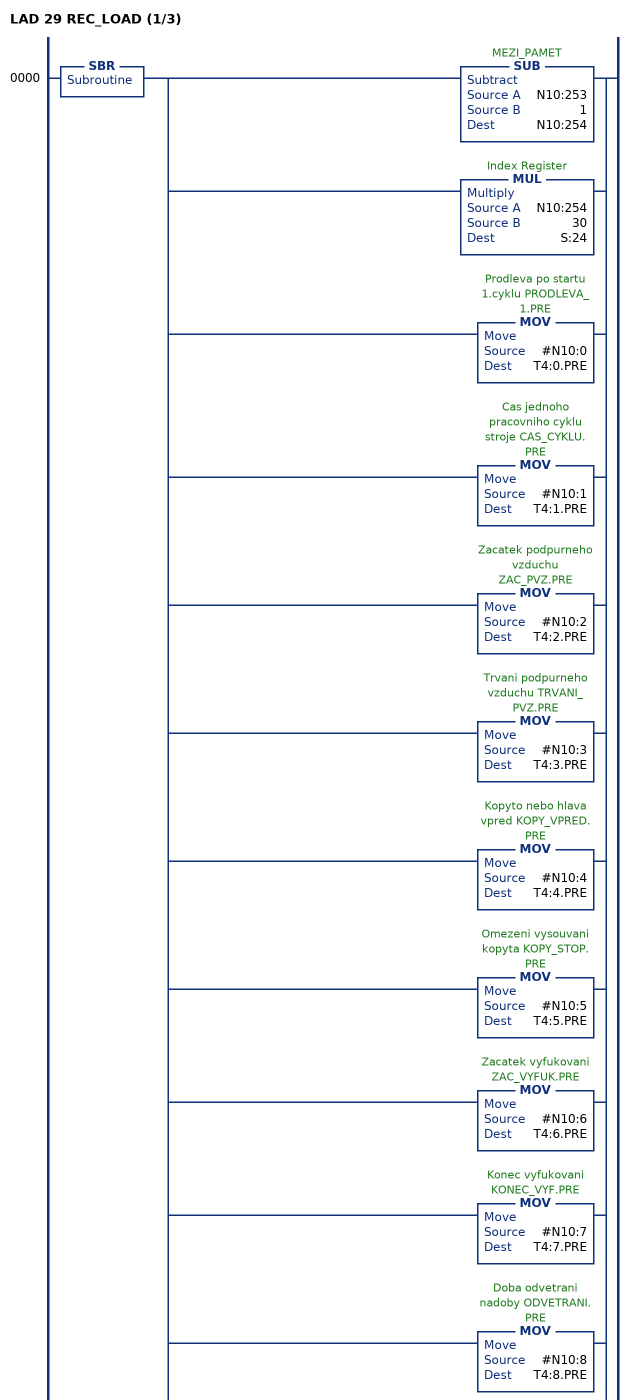
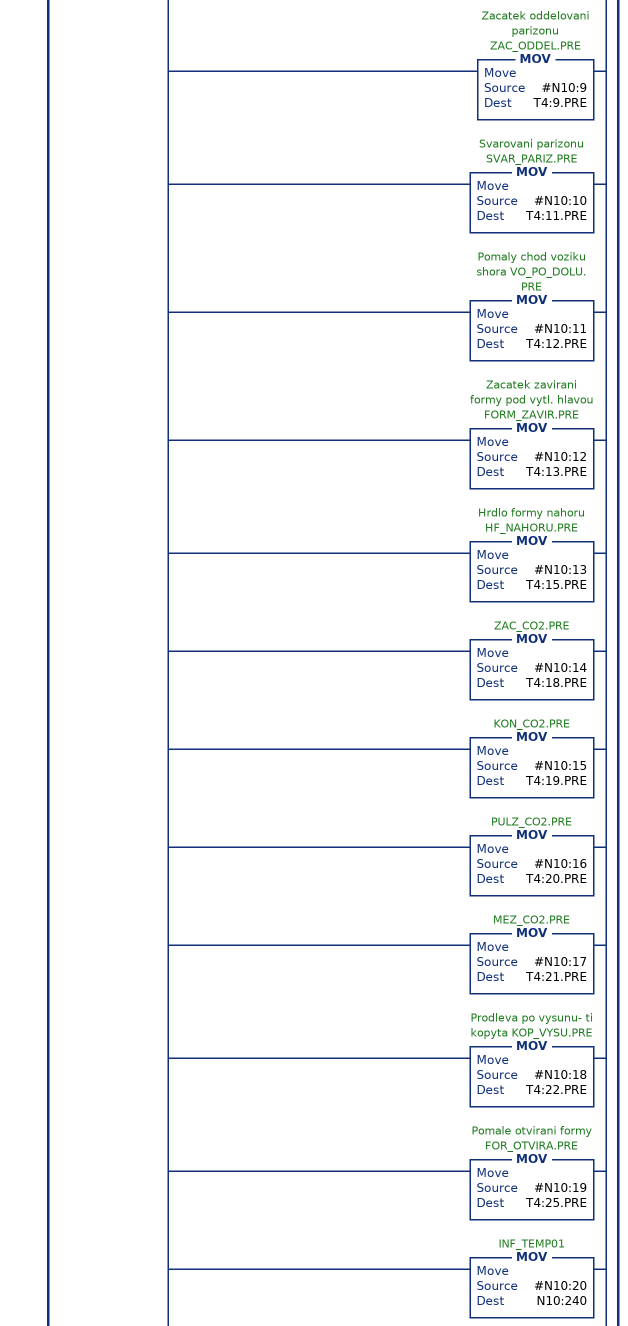
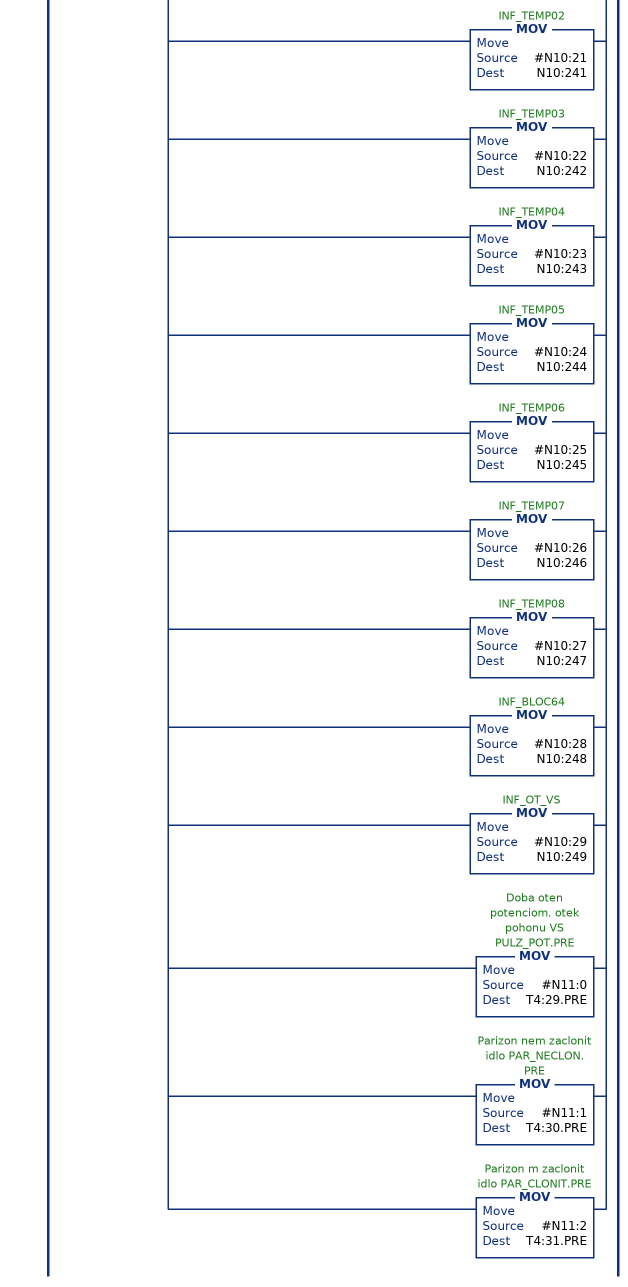
% Rung: 0 %
SOR SBR BST SUB N10:253 1 N10:254 NXB MUL N10:254 30 S:24 NXB MOV #N10:0 T4:0.PRE NXB MOV #N10:1 T4:1.PRE NXB MOV #N10:2 T4:2.PRE NXB MOV #N10:3 T4:3.PRE NXB MOV #N10:4 T4:4.PRE NXB MOV #N10:5 T4:5.PRE NXB MOV #N10:6 T4:6.PRE NXB MOV #N10:7 T4:7.PRE NXB MOV #N10:8 T4:8.PRE NXB MOV #N10:9 T4:9.PRE NXB MOV #N10:10 T4:11.PRE NXB MOV #N10:11 T4:12.PRE NXB MOV #N10:12 T4:13.PRE NXB MOV #N10:13 T4:15.PRE NXB MOV #N10:14 T4:18.PRE NXB MOV #N10:15 T4:19.PRE NXB MOV #N10:16 T4:20.PRE NXB MOV #N10:17 T4:21.PRE NXB MOV #N10:18 T4:22.PRE NXB MOV #N10:19 T4:25.PRE NXB MOV #N10:20 N10:240 NXB MOV #N10:21 N10:241 NXB MOV #N10:22 N10:242 NXB MOV #N10:23 N10:243 NXB MOV #N10:24 N10:244 NXB MOV #N10:25 N10:245 NXB MOV #N10:26 N10:246 NXB MOV #N10:27 N10:247 NXB MOV #N10:28 N10:248 NXB MOV #N10:29 N10:249 NXB MOV #N11:0 T4:29.PRE NXB MOV #N11:1 T4:30.PRE NXB MOV #N11:2 T4:31.PRE BND EOR
%   N10:253  REC_NO_PAR %
%   N10:254  MEZI_PAMET %
%   S:24  "Index Register" %
%   N10:0  REC_WORD00 %
%   T4:0  PRODLEVA_1  "Prodleva po startu 1.cyklu" %
%   N10:1  REC_WORD01 %
%   T4:1  CAS_CYKLU  "Cas jednoho pracovniho cyklu stroje" %
%   N10:2  REC_WORD02 %
%   T4:2  ZAC_PVZ  "Zacatek podpurneho vzduchu" %
%   N10:3  REC_WORD03 %
%   T4:3  TRVANI_PVZ  "Trvani podpurneho vzduchu" %
%   N10:4  REC_WORD04 %
%   T4:4  KOPY_VPRED  "Kopyto nebo hlava vpred" %
%   N10:5  REC_WORD05 %
%   T4:5  KOPY_STOP  "Omezeni vysouvani kopyta" %
%   N10:6  REC_WORD06 %
%   T4:6  ZAC_VYFUK  "Zacatek vyfukovani" %
%   N10:7  REC_WORD07 %
%   T4:7  KONEC_VYF  "Konec vyfukovani" %
%   N10:8  REC_WORD08 %
%   T4:8  ODVETRANI  "Doba odvetrani nadoby" %
%   N10:9  REC_WORD09 %
%   T4:9  ZAC_ODDEL  "Zacatek oddelovani parizonu" %
%   N10:10  REC_WORD10 %
%   T4:11  SVAR_PARIZ  "Svarovani parizonu" %
%   N10:11  REC_WORD11 %
%   T4:12  VO_PO_DOLU  "Pomaly chod voziku shora" %
%   N10:12  REC_WORD12 %
%   T4:13  FORM_ZAVIR  "Zacatek zavirani formy pod vytl. hlavou" %
%   N10:13  REC_WORD13 %
%   T4:15  HF_NAHORU  "Hrdlo formy nahoru" %
%   N10:14  REC_WORD14 %
%   T4:18  ZAC_CO2 %
%   N10:15  REC_WORD15 %
%   T4:19  KON_CO2 %
%   N10:16  REC_WORD16 %
%   T4:20  PULZ_CO2 %
%   N10:17  REC_WORD17 %
%   T4:21  MEZ_CO2 %
%   N10:18  REC_WORD18 %
%   T4:22  KOP_VYSU  "Prodleva po vysunu- ti kopyta" %
%   N10:19  REC_WORD19 %
%   T4:25  FOR_OTVIRA  "Pomale otvirani formy" %
%   N10:20  REC_WORD20 %
%   N10:240  INF_TEMP01 %
%   N10:21  REC_WORD21 %
%   N10:241  INF_TEMP02 %
%   N10:22  REC_WORD22 %
%   N10:242  INF_TEMP03 %
%   N10:23  REC_WORD23 %
%   N10:243  INF_TEMP04 %
%   N10:24  REC_WORD24 %
%   N10:244  INF_TEMP05 %
%   N10:25  REC_WORD25 %
%   N10:245  INF_TEMP06 %
%   N10:26  REC_WORD26 %
%   N10:246  INF_TEMP07 %
%   N10:27  REC_WORD27 %
%   N10:247  INF_TEMP08 %
%   N10:28  REC_WORD28 %
%   N10:248  INF_BLOC64 %
%   N10:29  REC_WORD29 %
%   N10:249  INF_OT_VS %
%   N11:0  REC_WORD30 %
%   T4:29  PULZ_POT  "Doba oten potenciom. otek pohonu VS" %
%   N11:1  REC_WORD31 %
%   T4:30  PAR_NECLON  "Parizon nem zaclonit idlo" %
%   N11:2  REC_WORD32 %
%   T4:31  PAR_CLONIT  "Parizon m zaclonit idlo" %

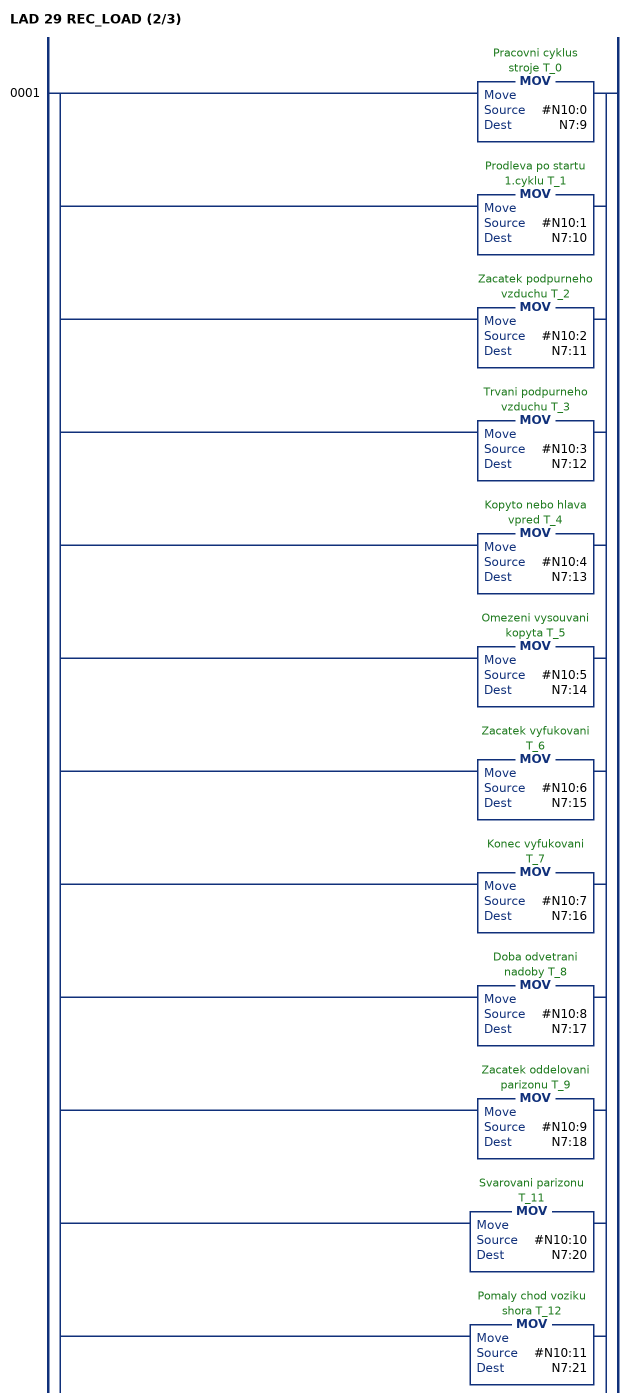

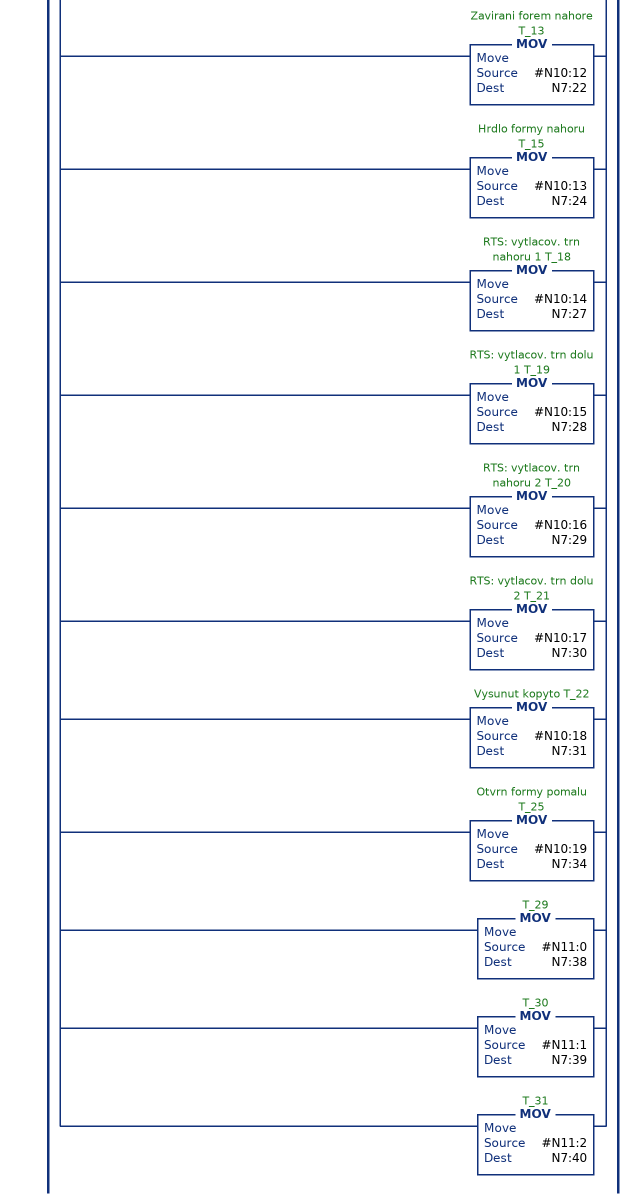
% Rung: 1 %
SOR BST MOV #N10:0 N7:9 NXB MOV #N10:1 N7:10 NXB MOV #N10:2 N7:11 NXB MOV #N10:3 N7:12 NXB MOV #N10:4 N7:13 NXB MOV #N10:5 N7:14 NXB MOV #N10:6 N7:15 NXB MOV #N10:7 N7:16 NXB MOV #N10:8 N7:17 NXB MOV #N10:9 N7:18 NXB MOV #N10:10 N7:20 NXB MOV #N10:11 N7:21 NXB MOV #N10:12 N7:22 NXB MOV #N10:13 N7:24 NXB MOV #N10:14 N7:27 NXB MOV #N10:15 N7:28 NXB MOV #N10:16 N7:29 NXB MOV #N10:17 N7:30 NXB MOV #N10:18 N7:31 NXB MOV #N10:19 N7:34 NXB MOV #N11:0 N7:38 NXB MOV #N11:1 N7:39 NXB MOV #N11:2 N7:40 BND EOR
%   N10:0  REC_WORD00 %
%   N7:9  T_0  "Pracovni cyklus stroje" %
%   N10:1  REC_WORD01 %
%   N7:10  T_1  "Prodleva po startu 1.cyklu" %
%   N10:2  REC_WORD02 %
%   N7:11  T_2  "Zacatek podpurneho vzduchu" %
%   N10:3  REC_WORD03 %
%   N7:12  T_3  "Trvani podpurneho vzduchu" %
%   N10:4  REC_WORD04 %
%   N7:13  T_4  "Kopyto nebo hlava vpred" %
%   N10:5  REC_WORD05 %
%   N7:14  T_5  "Omezeni vysouvani kopyta" %
%   N10:6  REC_WORD06 %
%   N7:15  T_6  "Zacatek vyfukovani" %
%   N10:7  REC_WORD07 %
%   N7:16  T_7  "Konec vyfukovani" %
%   N10:8  REC_WORD08 %
%   N7:17  T_8  "Doba odvetrani nadoby" %
%   N10:9  REC_WORD09 %
%   N7:18  T_9  "Zacatek oddelovani parizonu" %
%   N10:10  REC_WORD10 %
%   N7:20  T_11  "Svarovani parizonu" %
%   N10:11  REC_WORD11 %
%   N7:21  T_12  "Pomaly chod voziku shora" %
%   N10:12  REC_WORD12 %
%   N7:22  T_13  "Zavirani forem nahore" %
%   N10:13  REC_WORD13 %
%   N7:24  T_15  "Hrdlo formy nahoru" %
%   N10:14  REC_WORD14 %
%   N7:27  T_18  "RTS: vytlacov. trn nahoru 1" %
%   N10:15  REC_WORD15 %
%   N7:28  T_19  "RTS: vytlacov. trn dolu 1" %
%   N10:16  REC_WORD16 %
%   N7:29  T_20  "RTS: vytlacov. trn nahoru 2" %
%   N10:17  REC_WORD17 %
%   N7:30  T_21  "RTS: vytlacov. trn dolu 2" %
%   N10:18  REC_WORD18 %
%   N7:31  T_22  "Vysunut kopyto" %
%   N10:19  REC_WORD19 %
%   N7:34  T_25  "Otvrn formy pomalu" %
%   N11:0  REC_WORD30 %
%   N7:38  T_29 %
%   N11:1  REC_WORD31 %
%   N7:39  T_30 %
%   N11:2  REC_WORD32 %
%   N7:40  T_31 %

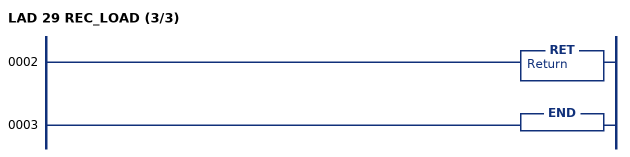
% Rung: 2 %
SOR RET EOR
% Rung: 3 %
SOR END EOR

LADDER 30 "REG_TEPLOT"
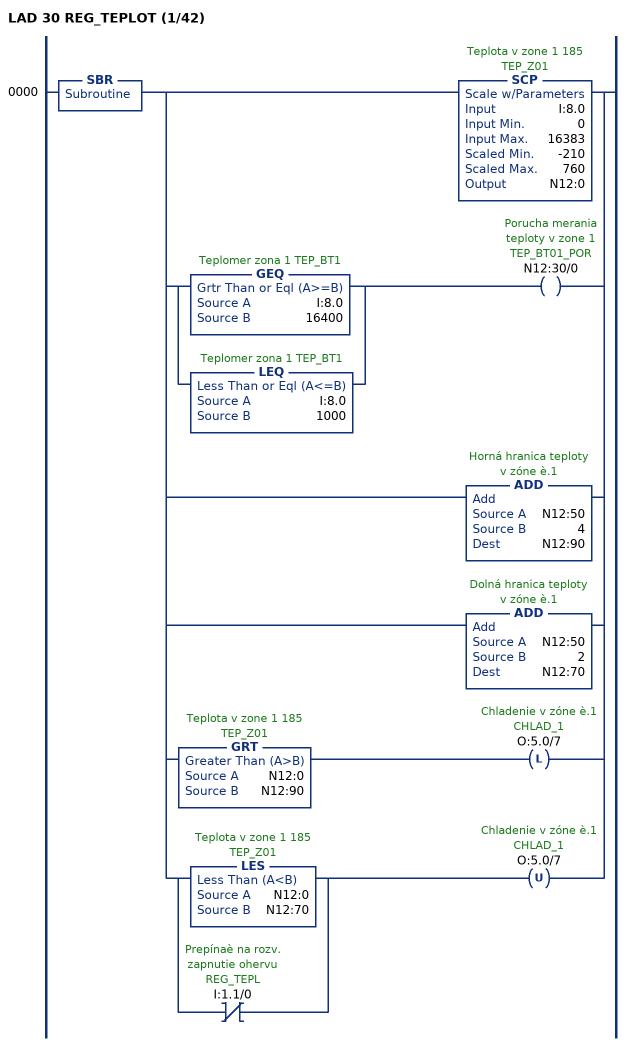
% Rung: 0 %
SOR SBR BST SCP I:8.0 0 16383 -210 760 N12:0 NXB BST GEQ I:8.0 16400 NXB LEQ I:8.0 1000 BND OTE N12:30/0 NXB ADD N12:50 4 N12:90 NXB ADD N12:50 2 N12:70 NXB GRT N12:0 N12:90 OTL O:5.0/7 NXB BST LES N12:0 N12:70 NXB XIO I:1.1/0 BND OTU O:5.0/7 BND EOR
%   I:8.0  TEP_BT1  "Teplomer zona 1" %
%   N12:0  TEP_Z01  "Teplota v zone 1 185" %
%   N12:30/0  TEP_BT01_POR  "Porucha merania teploty v zone 1" %
%   N12:50  "Žiadaná teplota v zóne è.1" %
%   N12:90  "Horná hranica teploty v zóne è.1" %
%   N12:70  "Dolná hranica teploty v zóne è.1" %
%   O:5.0/7  CHLAD_1  "Chladenie v zóne è.1" %
%   I:1.1/0  REG_TEPL  "Prepínaè na rozv. zapnutie ohervu" %

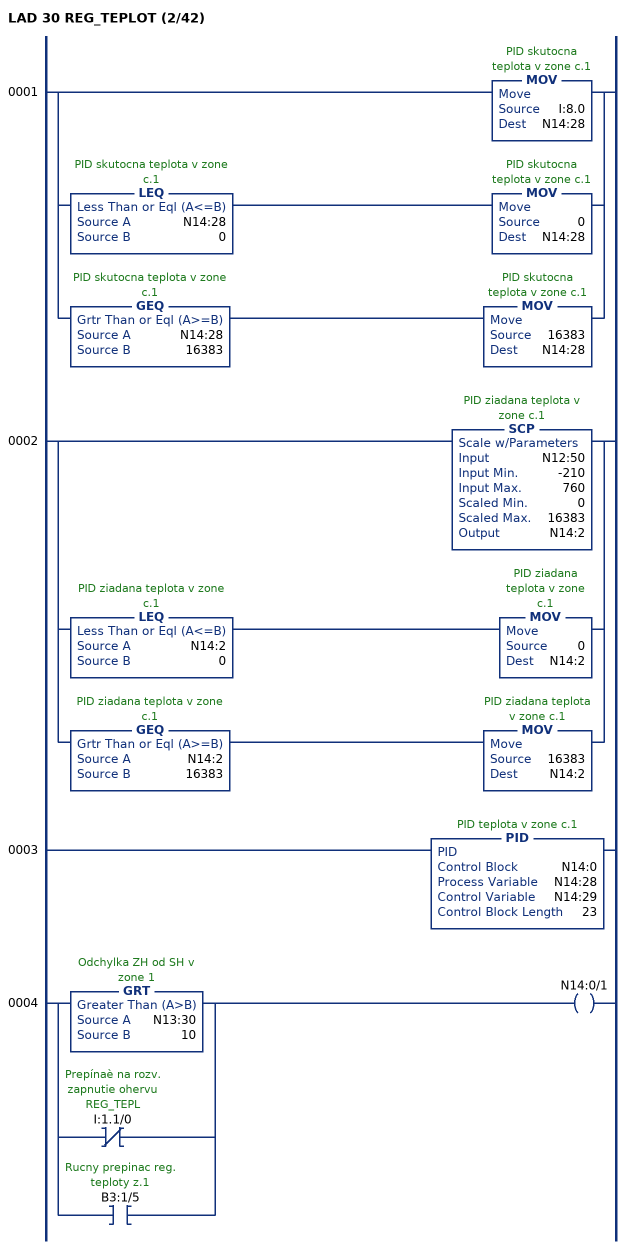
% Rung: 1 %
SOR BST MOV I:8.0 N14:28 NXB LEQ N14:28 0 MOV 0 N14:28 NXB GEQ N14:28 16383 MOV 16383 N14:28 BND EOR
%   I:8.0  TEP_BT1  "Teplomer zona 1" %
%   N14:28  "PID skutocna teplota v zone c.1" %
% Rung: 2 %
SOR BST SCP N12:50 -210 760 0 16383 N14:2 NXB LEQ N14:2 0 MOV 0 N14:2 NXB GEQ N14:2 16383 MOV 16383 N14:2 BND EOR
%   N12:50  "Žiadaná teplota v zóne è.1" %
%   N14:2  "PID ziadana teplota v zone c.1" %
% Rung: 3 %
SOR PID N14:0 N14:28 N14:29 23 EOR
%   N14:0  "PID teplota v zone c.1" %
%   N14:28  "PID skutocna teplota v zone c.1" %
% Rung: 4 %
SOR BST GRT N13:30 10 NXB XIO I:1.1/0 NXB XIC B3:1/5 BND OTE N14:0/1 EOR
%   N13:30  "Odchylka ZH od SH v zone 1" %
%   I:1.1/0  REG_TEPL  "Prepínaè na rozv. zapnutie ohervu" %
%   B3:1/5  "Rucny prepinac reg. teploty z.1" %

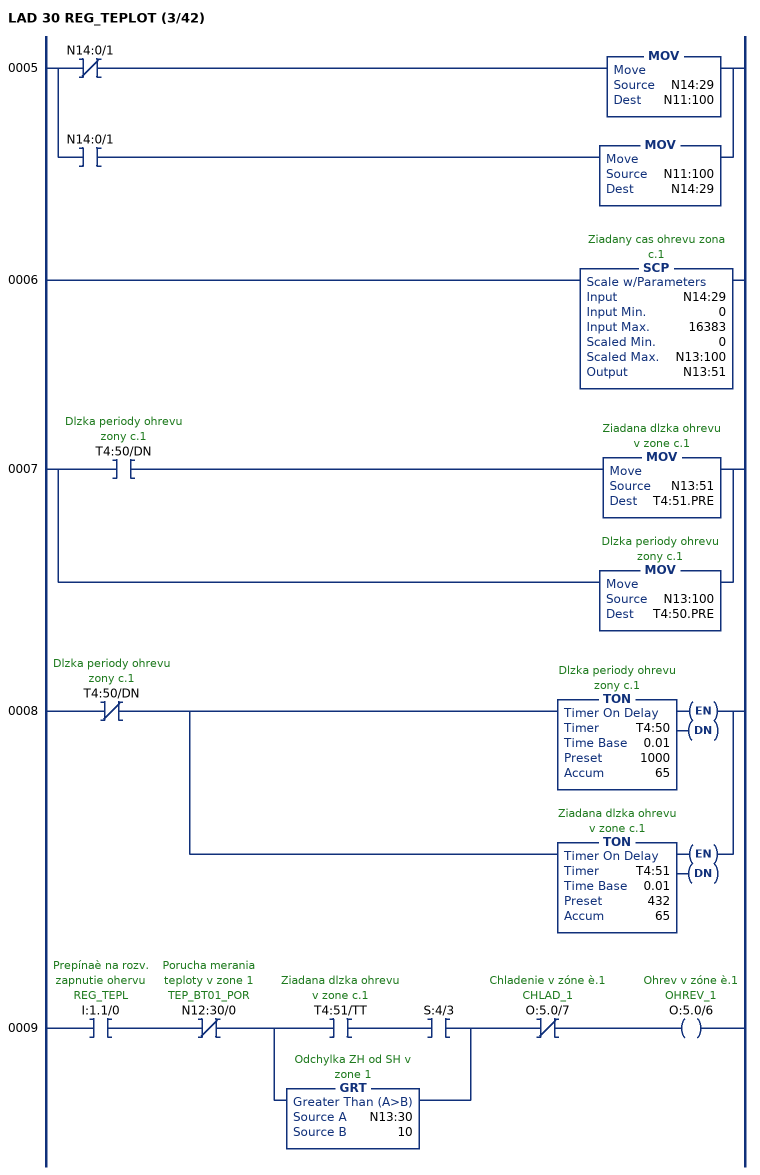
% Rung: 5 %
SOR BST XIO N14:0/1 MOV N14:29 N11:100 NXB XIC N14:0/1 MOV N11:100 N14:29 BND EOR
% Rung: 6 %
SOR SCP N14:29 0 16383 0 N13:100 N13:51 EOR
%   N13:51  "Ziadany cas ohrevu zona c.1" %
% Rung: 7 %
SOR BST XIC T4:50/DN MOV N13:51 T4:51.PRE NXB MOV N13:100 T4:50.PRE BND EOR
%   T4:50  "Dlzka periody ohrevu zony c.1" %
%   N13:51  "Ziadany cas ohrevu zona c.1" %
%   T4:51  "Ziadana dlzka ohrevu v zone c.1" %
% Rung: 8 %
SOR XIO T4:50/DN BST TON T4:50 0.01 1000 65 NXB TON T4:51 0.01 432 65 BND EOR
%   T4:50  "Dlzka periody ohrevu zony c.1" %
%   T4:51  "Ziadana dlzka ohrevu v zone c.1" %
% Rung: 9 %
SOR XIC I:1.1/0 XIO N12:30/0 BST XIC T4:51/TT XIC S:4/3 NXB GRT N13:30 10 BND XIO O:5.0/7 OTE O:5.0/6 EOR
%   I:1.1/0  REG_TEPL  "Prepínaè na rozv. zapnutie ohervu" %
%   N12:30/0  TEP_BT01_POR  "Porucha merania teploty v zone 1" %
%   T4:51  "Ziadana dlzka ohrevu v zone c.1" %
%   N13:30  "Odchylka ZH od SH v zone 1" %
%   O:5.0/7  CHLAD_1  "Chladenie v zóne è.1" %
%   O:5.0/6  OHREV_1  "Ohrev v zóne è.1" %

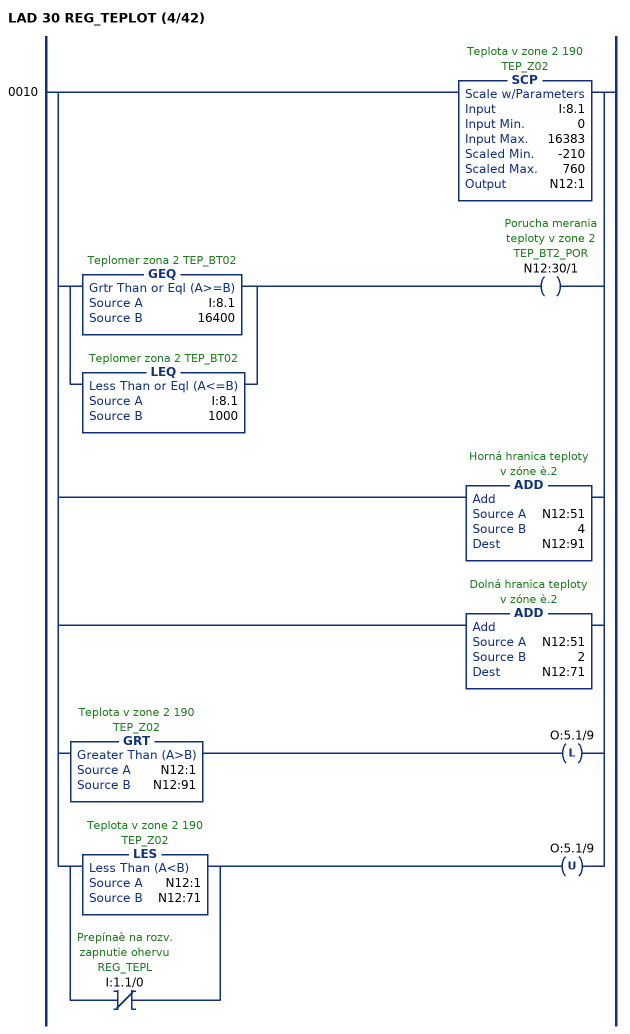
% Rung: 10 %
SOR BST SCP I:8.1 0 16383 -210 760 N12:1 NXB BST GEQ I:8.1 16400 NXB LEQ I:8.1 1000 BND OTE N12:30/1 NXB ADD N12:51 4 N12:91 NXB ADD N12:51 2 N12:71 NXB GRT N12:1 N12:91 OTL O:5.1/9 NXB BST LES N12:1 N12:71 NXB XIO I:1.1/0 BND OTU O:5.1/9 BND EOR
%   I:8.1  TEP_BT02  "Teplomer zona 2" %
%   N12:1  TEP_Z02  "Teplota v zone 2 190" %
%   N12:30/1  TEP_BT2_POR  "Porucha merania teploty v zone 2" %
%   N12:51  "Žiadaná teplota v zóne è.2" %
%   N12:91  "Horná hranica teploty v zóne è.2" %
%   N12:71  "Dolná hranica teploty v zóne è.2" %
%   I:1.1/0  REG_TEPL  "Prepínaè na rozv. zapnutie ohervu" %

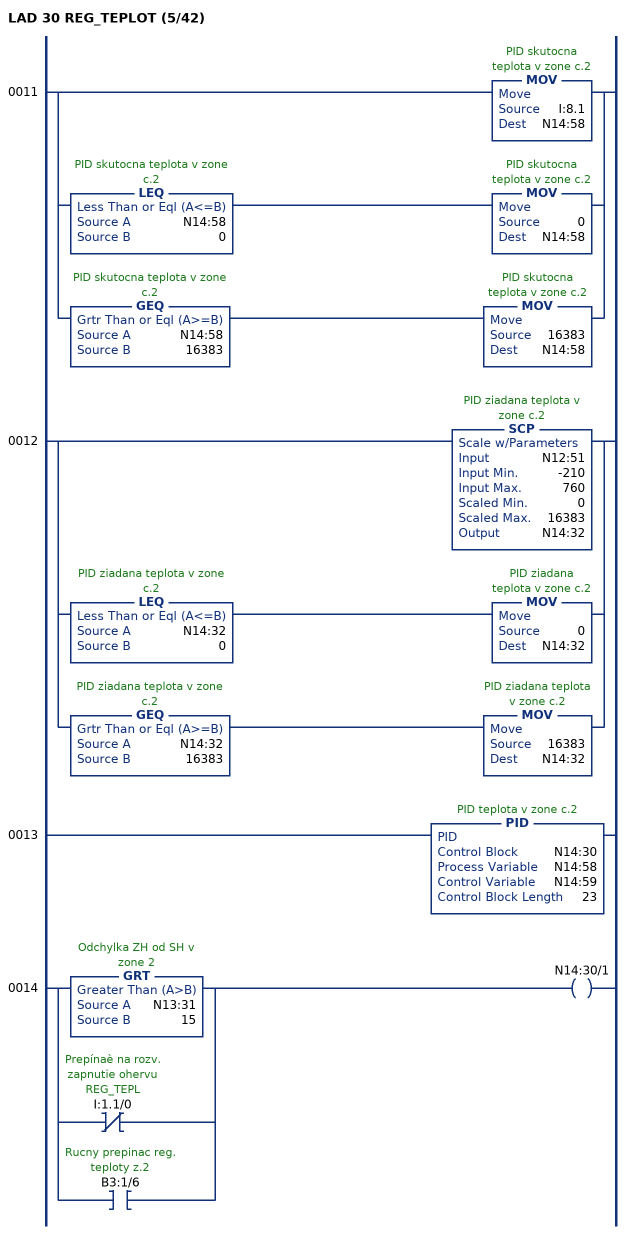
% Rung: 11 %
SOR BST MOV I:8.1 N14:58 NXB LEQ N14:58 0 MOV 0 N14:58 NXB GEQ N14:58 16383 MOV 16383 N14:58 BND EOR
%   I:8.1  TEP_BT02  "Teplomer zona 2" %
%   N14:58  "PID skutocna teplota v zone c.2" %
% Rung: 12 %
SOR BST SCP N12:51 -210 760 0 16383 N14:32 NXB LEQ N14:32 0 MOV 0 N14:32 NXB GEQ N14:32 16383 MOV 16383 N14:32 BND EOR
%   N12:51  "Žiadaná teplota v zóne è.2" %
%   N14:32  "PID ziadana teplota v zone c.2" %
% Rung: 13 %
SOR PID N14:30 N14:58 N14:59 23 EOR
%   N14:30  "PID teplota v zone c.2" %
%   N14:58  "PID skutocna teplota v zone c.2" %
% Rung: 14 %
SOR BST GRT N13:31 15 NXB XIO I:1.1/0 NXB XIC B3:1/6 BND OTE N14:30/1 EOR
%   N13:31  "Odchylka ZH od SH v zone 2" %
%   I:1.1/0  REG_TEPL  "Prepínaè na rozv. zapnutie ohervu" %
%   B3:1/6  "Rucny prepinac reg. teploty z.2" %

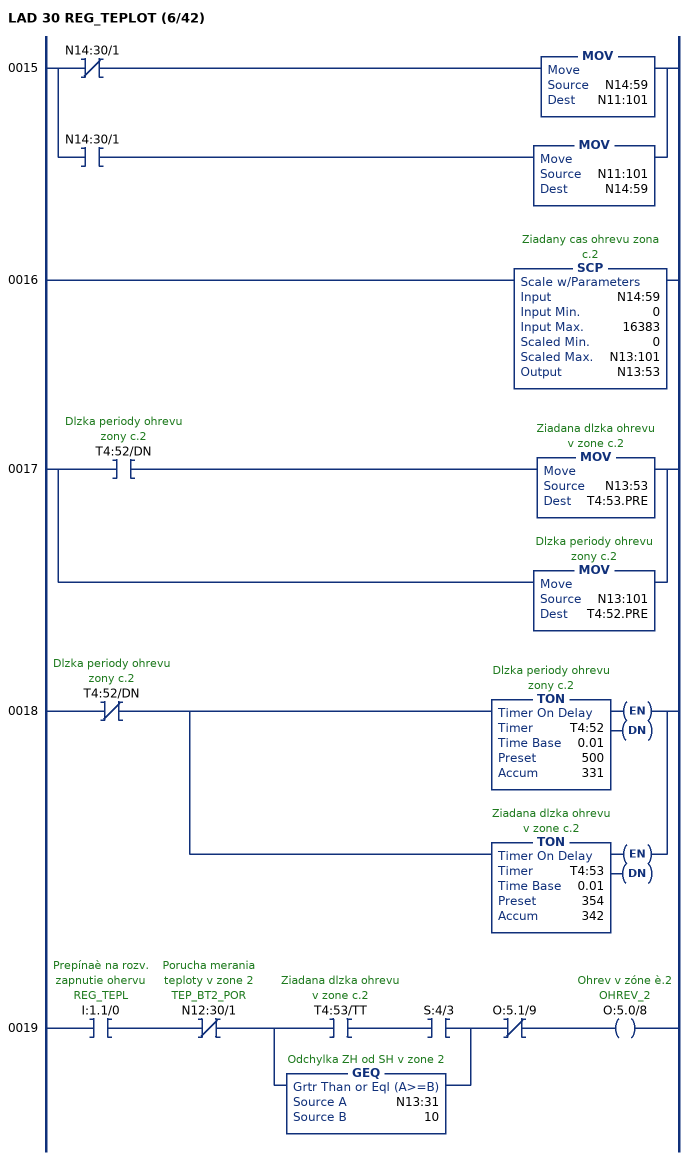
% Rung: 15 %
SOR BST XIO N14:30/1 MOV N14:59 N11:101 NXB XIC N14:30/1 MOV N11:101 N14:59 BND EOR
% Rung: 16 %
SOR SCP N14:59 0 16383 0 N13:101 N13:53 EOR
%   N13:53  "Ziadany cas ohrevu zona c.2" %
% Rung: 17 %
SOR BST XIC T4:52/DN MOV N13:53 T4:53.PRE NXB MOV N13:101 T4:52.PRE BND EOR
%   T4:52  "Dlzka periody ohrevu zony c.2" %
%   N13:53  "Ziadany cas ohrevu zona c.2" %
%   T4:53  "Ziadana dlzka ohrevu v zone c.2" %
% Rung: 18 %
SOR XIO T4:52/DN BST TON T4:52 0.01 500 331 NXB TON T4:53 0.01 354 342 BND EOR
%   T4:52  "Dlzka periody ohrevu zony c.2" %
%   T4:53  "Ziadana dlzka ohrevu v zone c.2" %
% Rung: 19 %
SOR XIC I:1.1/0 XIO N12:30/1 BST XIC T4:53/TT XIC S:4/3 NXB GEQ N13:31 10 BND XIO O:5.1/9 OTE O:5.0/8 EOR
%   I:1.1/0  REG_TEPL  "Prepínaè na rozv. zapnutie ohervu" %
%   N12:30/1  TEP_BT2_POR  "Porucha merania teploty v zone 2" %
%   T4:53  "Ziadana dlzka ohrevu v zone c.2" %
%   N13:31  "Odchylka ZH od SH v zone 2" %
%   O:5.0/8  OHREV_2  "Ohrev v zóne è.2" %

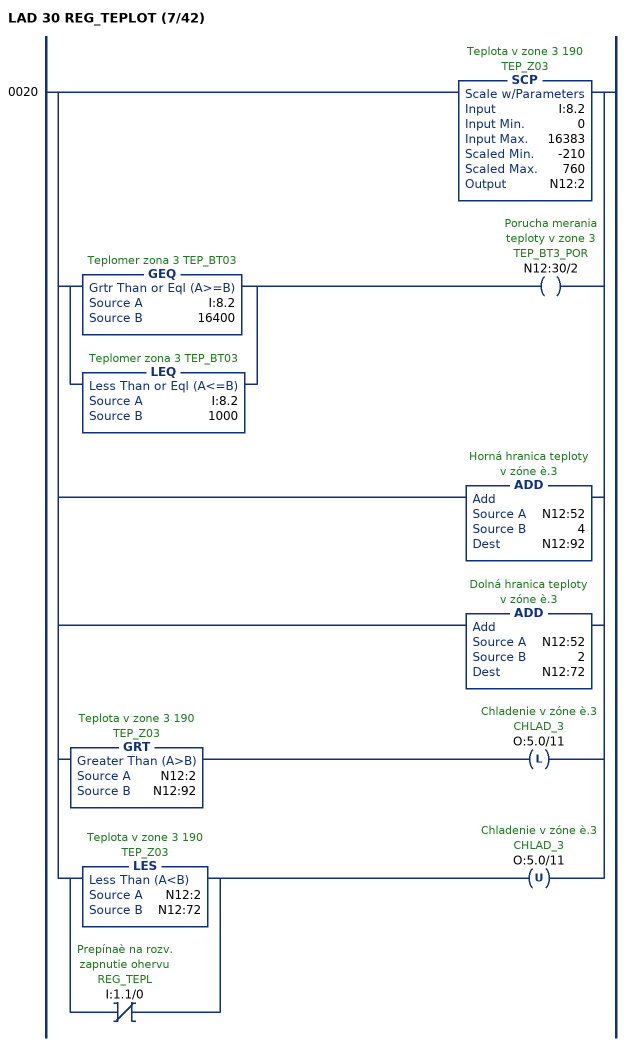
% Rung: 20 %
SOR BST SCP I:8.2 0 16383 -210 760 N12:2 NXB BST GEQ I:8.2 16400 NXB LEQ I:8.2 1000 BND OTE N12:30/2 NXB ADD N12:52 4 N12:92 NXB ADD N12:52 2 N12:72 NXB GRT N12:2 N12:92 OTL O:5.0/11 NXB BST LES N12:2 N12:72 NXB XIO I:1.1/0 BND OTU O:5.0/11 BND EOR
%   I:8.2  TEP_BT03  "Teplomer zona 3" %
%   N12:2  TEP_Z03  "Teplota v zone 3 190" %
%   N12:30/2  TEP_BT3_POR  "Porucha merania teploty v zone 3" %
%   N12:52  "Žiadaná teplota v zóne è.3" %
%   N12:92  "Horná hranica teploty v zóne è.3" %
%   N12:72  "Dolná hranica teploty v zóne è.3" %
%   O:5.0/11  CHLAD_3  "Chladenie v zóne è.3" %
%   I:1.1/0  REG_TEPL  "Prepínaè na rozv. zapnutie ohervu" %

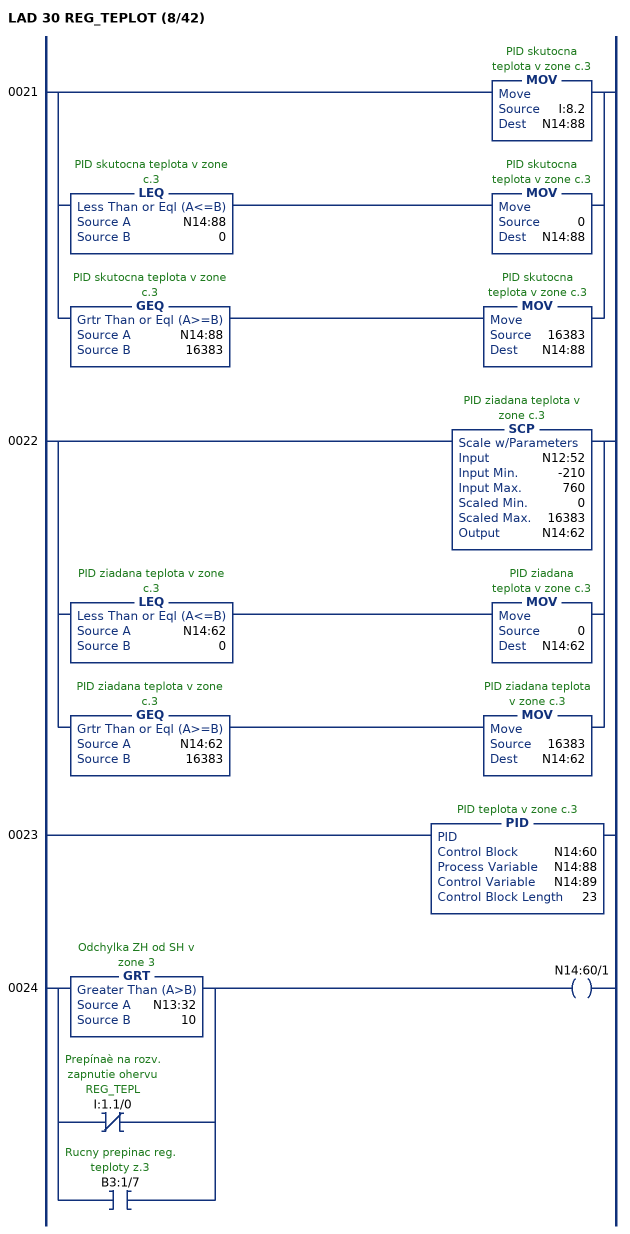
% Rung: 21 %
SOR BST MOV I:8.2 N14:88 NXB LEQ N14:88 0 MOV 0 N14:88 NXB GEQ N14:88 16383 MOV 16383 N14:88 BND EOR
%   I:8.2  TEP_BT03  "Teplomer zona 3" %
%   N14:88  "PID skutocna teplota v zone c.3" %
% Rung: 22 %
SOR BST SCP N12:52 -210 760 0 16383 N14:62 NXB LEQ N14:62 0 MOV 0 N14:62 NXB GEQ N14:62 16383 MOV 16383 N14:62 BND EOR
%   N12:52  "Žiadaná teplota v zóne è.3" %
%   N14:62  "PID ziadana teplota v zone c.3" %
% Rung: 23 %
SOR PID N14:60 N14:88 N14:89 23 EOR
%   N14:60  "PID teplota v zone c.3" %
%   N14:88  "PID skutocna teplota v zone c.3" %
% Rung: 24 %
SOR BST GRT N13:32 10 NXB XIO I:1.1/0 NXB XIC B3:1/7 BND OTE N14:60/1 EOR
%   N13:32  "Odchylka ZH od SH v zone 3" %
%   I:1.1/0  REG_TEPL  "Prepínaè na rozv. zapnutie ohervu" %
%   B3:1/7  "Rucny prepinac reg. teploty z.3" %

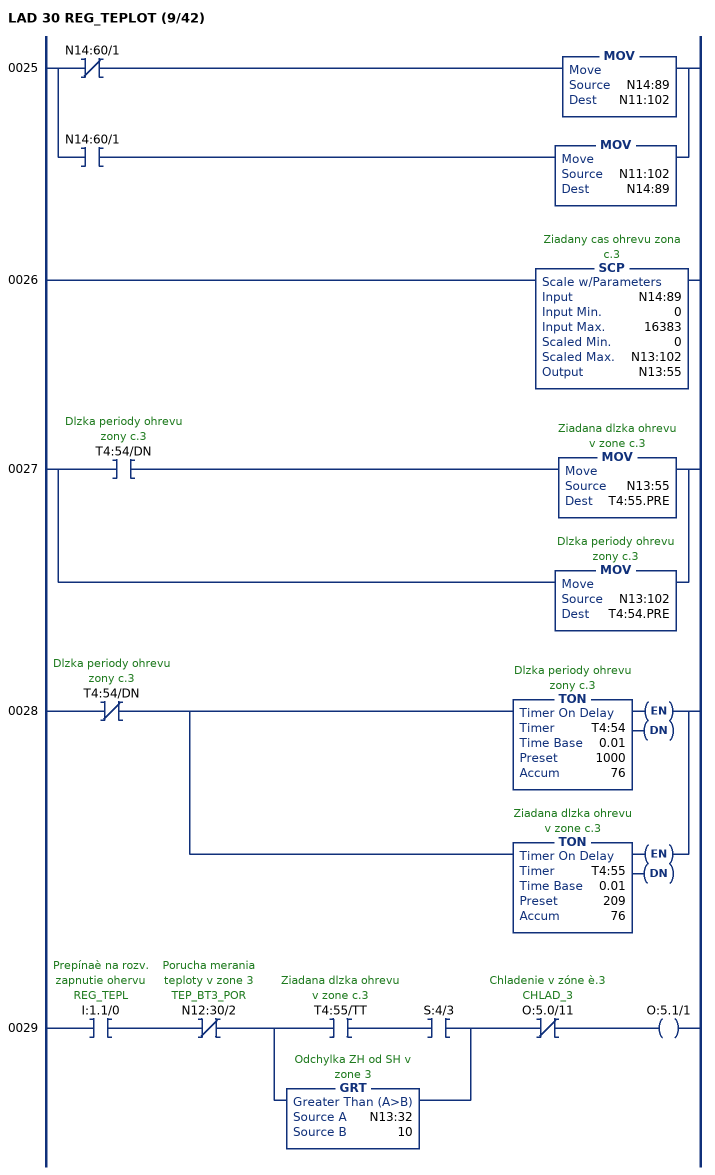
% Rung: 25 %
SOR BST XIO N14:60/1 MOV N14:89 N11:102 NXB XIC N14:60/1 MOV N11:102 N14:89 BND EOR
% Rung: 26 %
SOR SCP N14:89 0 16383 0 N13:102 N13:55 EOR
%   N13:55  "Ziadany cas ohrevu zona c.3" %
% Rung: 27 %
SOR BST XIC T4:54/DN MOV N13:55 T4:55.PRE NXB MOV N13:102 T4:54.PRE BND EOR
%   T4:54  "Dlzka periody ohrevu zony c.3" %
%   N13:55  "Ziadany cas ohrevu zona c.3" %
%   T4:55  "Ziadana dlzka ohrevu v zone c.3" %
% Rung: 28 %
SOR XIO T4:54/DN BST TON T4:54 0.01 1000 76 NXB TON T4:55 0.01 209 76 BND EOR
%   T4:54  "Dlzka periody ohrevu zony c.3" %
%   T4:55  "Ziadana dlzka ohrevu v zone c.3" %
% Rung: 29 %
SOR XIC I:1.1/0 XIO N12:30/2 BST XIC T4:55/TT XIC S:4/3 NXB GRT N13:32 10 BND XIO O:5.0/11 OTE O:5.1/1 EOR
%   I:1.1/0  REG_TEPL  "Prepínaè na rozv. zapnutie ohervu" %
%   N12:30/2  TEP_BT3_POR  "Porucha merania teploty v zone 3" %
%   T4:55  "Ziadana dlzka ohrevu v zone c.3" %
%   N13:32  "Odchylka ZH od SH v zone 3" %
%   O:5.0/11  CHLAD_3  "Chladenie v zóne è.3" %

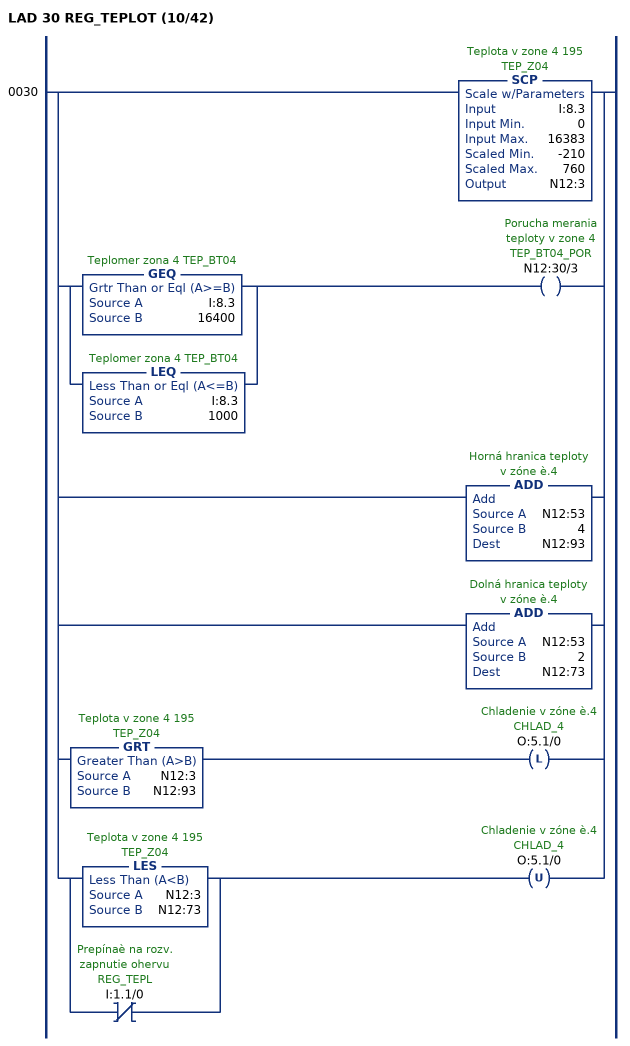
% Rung: 30 %
SOR BST SCP I:8.3 0 16383 -210 760 N12:3 NXB BST GEQ I:8.3 16400 NXB LEQ I:8.3 1000 BND OTE N12:30/3 NXB ADD N12:53 4 N12:93 NXB ADD N12:53 2 N12:73 NXB GRT N12:3 N12:93 OTL O:5.1/0 NXB BST LES N12:3 N12:73 NXB XIO I:1.1/0 BND OTU O:5.1/0 BND EOR
%   I:8.3  TEP_BT04  "Teplomer zona 4" %
%   N12:3  TEP_Z04  "Teplota v zone 4 195" %
%   N12:30/3  TEP_BT04_POR  "Porucha merania teploty v zone 4" %
%   N12:53  "Žiadaná teplota v zóne è.4" %
%   N12:93  "Horná hranica teploty v zóne è.4" %
%   N12:73  "Dolná hranica teploty v zóne è.4" %
%   O:5.1/0  CHLAD_4  "Chladenie v zóne è.4" %
%   I:1.1/0  REG_TEPL  "Prepínaè na rozv. zapnutie ohervu" %

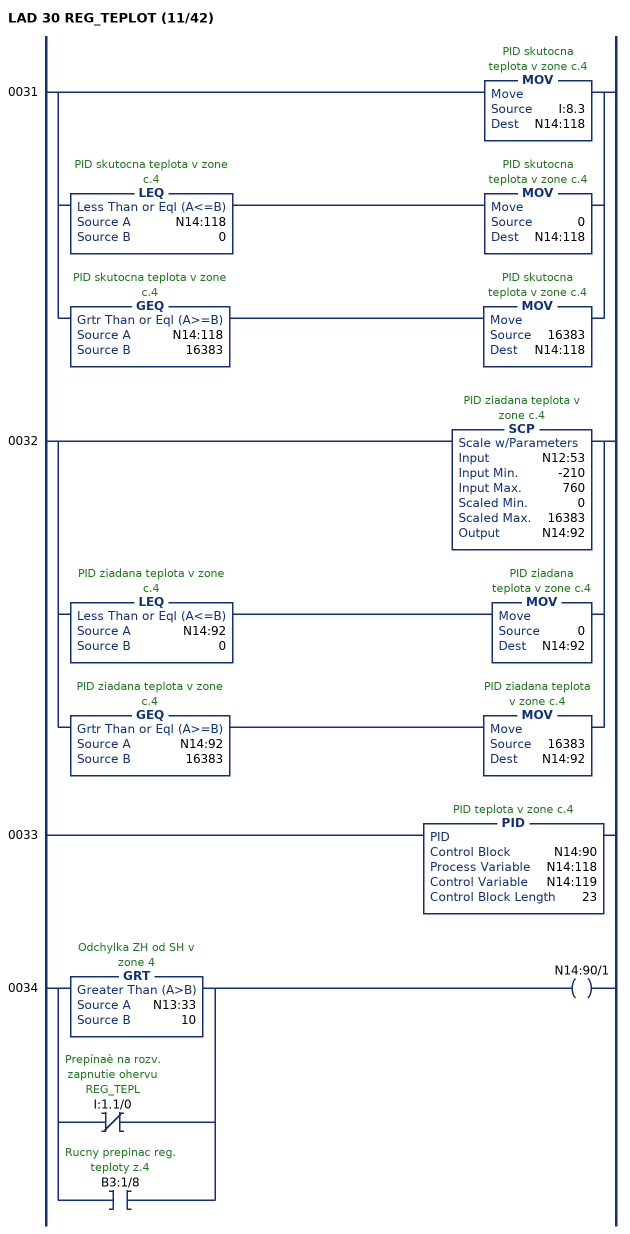
% Rung: 31 %
SOR BST MOV I:8.3 N14:118 NXB LEQ N14:118 0 MOV 0 N14:118 NXB GEQ N14:118 16383 MOV 16383 N14:118 BND EOR
%   I:8.3  TEP_BT04  "Teplomer zona 4" %
%   N14:118  "PID skutocna teplota v zone c.4" %
% Rung: 32 %
SOR BST SCP N12:53 -210 760 0 16383 N14:92 NXB LEQ N14:92 0 MOV 0 N14:92 NXB GEQ N14:92 16383 MOV 16383 N14:92 BND EOR
%   N12:53  "Žiadaná teplota v zóne è.4" %
%   N14:92  "PID ziadana teplota v zone c.4" %
% Rung: 33 %
SOR PID N14:90 N14:118 N14:119 23 EOR
%   N14:90  "PID teplota v zone c.4" %
%   N14:118  "PID skutocna teplota v zone c.4" %
% Rung: 34 %
SOR BST GRT N13:33 10 NXB XIO I:1.1/0 NXB XIC B3:1/8 BND OTE N14:90/1 EOR
%   N13:33  "Odchylka ZH od SH v zone 4" %
%   I:1.1/0  REG_TEPL  "Prepínaè na rozv. zapnutie ohervu" %
%   B3:1/8  "Rucny prepinac reg. teploty z.4" %

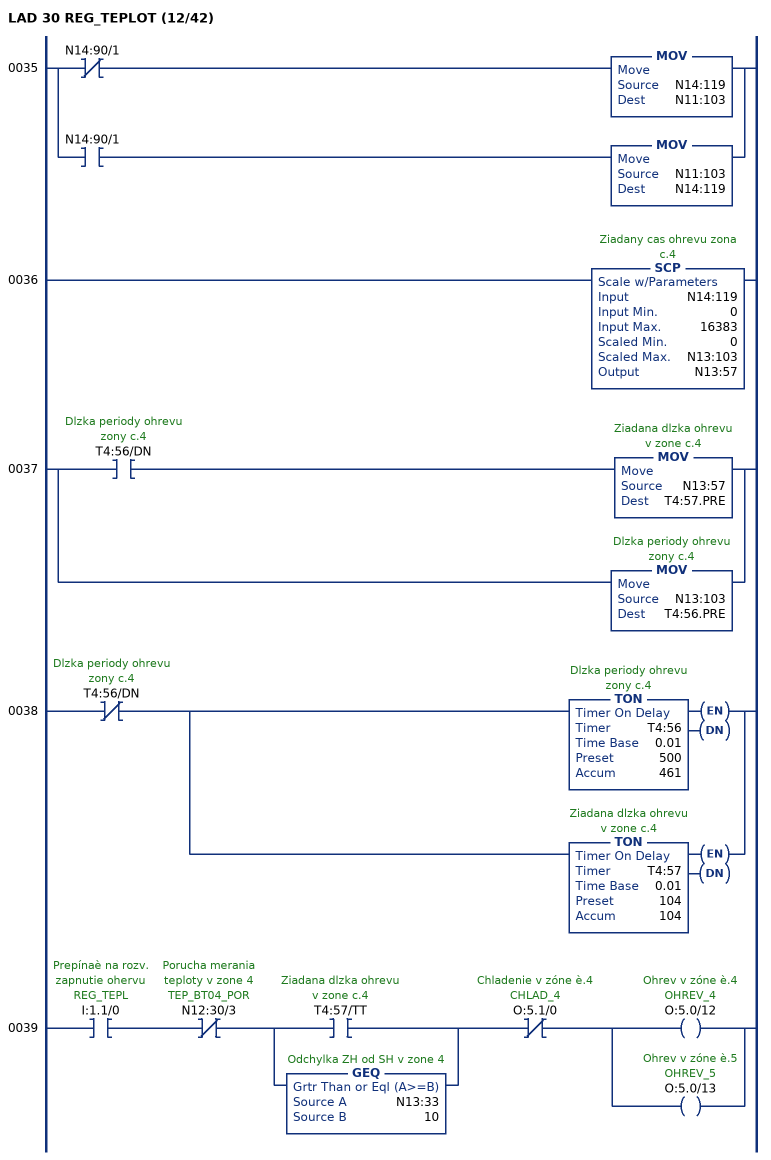
% Rung: 35 %
SOR BST XIO N14:90/1 MOV N14:119 N11:103 NXB XIC N14:90/1 MOV N11:103 N14:119 BND EOR
% Rung: 36 %
SOR SCP N14:119 0 16383 0 N13:103 N13:57 EOR
%   N13:57  "Ziadany cas ohrevu zona c.4" %
% Rung: 37 %
SOR BST XIC T4:56/DN MOV N13:57 T4:57.PRE NXB MOV N13:103 T4:56.PRE BND EOR
%   T4:56  "Dlzka periody ohrevu zony c.4" %
%   N13:57  "Ziadany cas ohrevu zona c.4" %
%   T4:57  "Ziadana dlzka ohrevu v zone c.4" %
% Rung: 38 %
SOR XIO T4:56/DN BST TON T4:56 0.01 500 461 NXB TON T4:57 0.01 104 104 BND EOR
%   T4:56  "Dlzka periody ohrevu zony c.4" %
%   T4:57  "Ziadana dlzka ohrevu v zone c.4" %
% Rung: 39 %
SOR XIC I:1.1/0 XIO N12:30/3 BST XIC T4:57/TT NXB GEQ N13:33 10 BND XIO O:5.1/0 BST OTE O:5.0/12 NXB OTE O:5.0/13 BND EOR
%   I:1.1/0  REG_TEPL  "Prepínaè na rozv. zapnutie ohervu" %
%   N12:30/3  TEP_BT04_POR  "Porucha merania teploty v zone 4" %
%   T4:57  "Ziadana dlzka ohrevu v zone c.4" %
%   N13:33  "Odchylka ZH od SH v zone 4" %
%   O:5.1/0  CHLAD_4  "Chladenie v zóne è.4" %
%   O:5.0/12  OHREV_4  "Ohrev v zóne è.4" %
%   O:5.0/13  OHREV_5  "Ohrev v zóne è.5" %

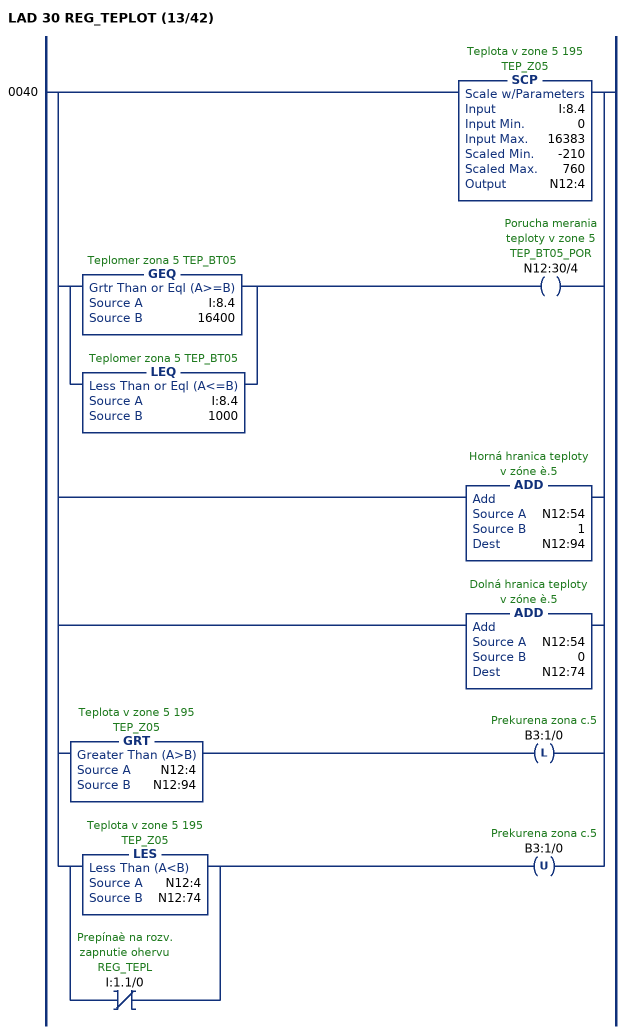
% Rung: 40 %
SOR BST SCP I:8.4 0 16383 -210 760 N12:4 NXB BST GEQ I:8.4 16400 NXB LEQ I:8.4 1000 BND OTE N12:30/4 NXB ADD N12:54 1 N12:94 NXB ADD N12:54 0 N12:74 NXB GRT N12:4 N12:94 OTL B3:1/0 NXB BST LES N12:4 N12:74 NXB XIO I:1.1/0 BND OTU B3:1/0 BND EOR
%   I:8.4  TEP_BT05  "Teplomer zona 5" %
%   N12:4  TEP_Z05  "Teplota v zone 5 195" %
%   N12:30/4  TEP_BT05_POR  "Porucha merania teploty v zone 5" %
%   N12:54  "Žiadaná teplota v zóne è.5" %
%   N12:94  "Horná hranica teploty v zóne è.5" %
%   N12:74  "Dolná hranica teploty v zóne è.5" %
%   B3:1/0  "Prekurena zona c.5" %
%   I:1.1/0  REG_TEPL  "Prepínaè na rozv. zapnutie ohervu" %

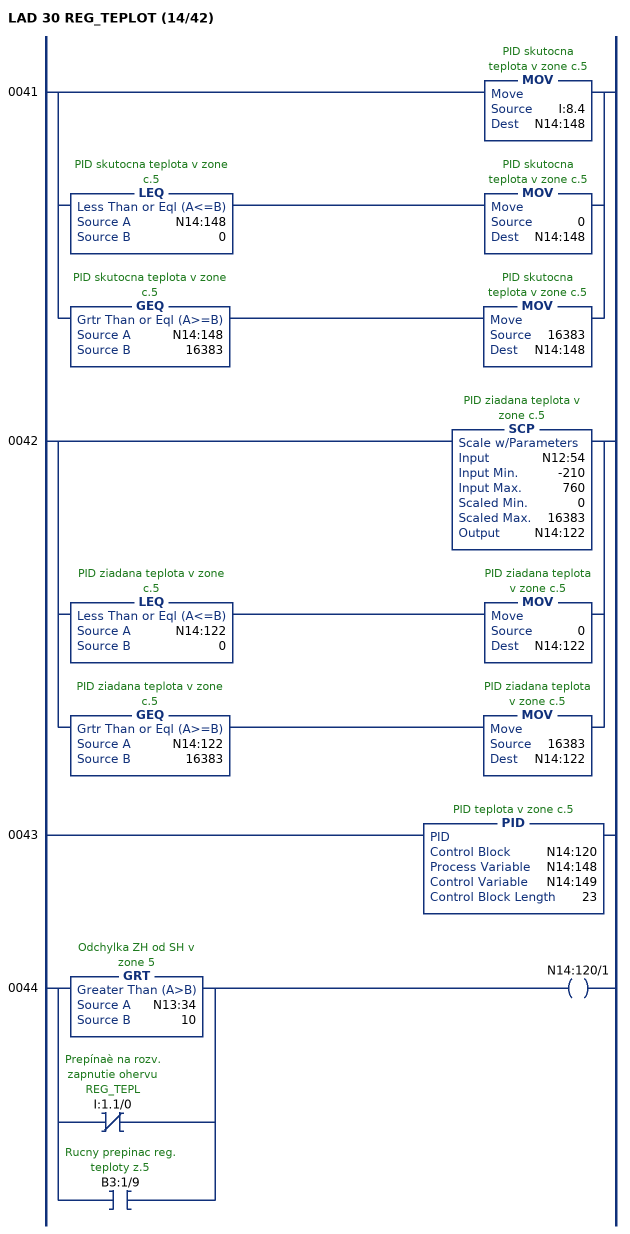
% Rung: 41 %
SOR BST MOV I:8.4 N14:148 NXB LEQ N14:148 0 MOV 0 N14:148 NXB GEQ N14:148 16383 MOV 16383 N14:148 BND EOR
%   I:8.4  TEP_BT05  "Teplomer zona 5" %
%   N14:148  "PID skutocna teplota v zone c.5" %
% Rung: 42 %
SOR BST SCP N12:54 -210 760 0 16383 N14:122 NXB LEQ N14:122 0 MOV 0 N14:122 NXB GEQ N14:122 16383 MOV 16383 N14:122 BND EOR
%   N12:54  "Žiadaná teplota v zóne è.5" %
%   N14:122  "PID ziadana teplota v zone c.5" %
% Rung: 43 %
SOR PID N14:120 N14:148 N14:149 23 EOR
%   N14:120  "PID teplota v zone c.5" %
%   N14:148  "PID skutocna teplota v zone c.5" %
% Rung: 44 %
SOR BST GRT N13:34 10 NXB XIO I:1.1/0 NXB XIC B3:1/9 BND OTE N14:120/1 EOR
%   N13:34  "Odchylka ZH od SH v zone 5" %
%   I:1.1/0  REG_TEPL  "Prepínaè na rozv. zapnutie ohervu" %
%   B3:1/9  "Rucny prepinac reg. teploty z.5" %

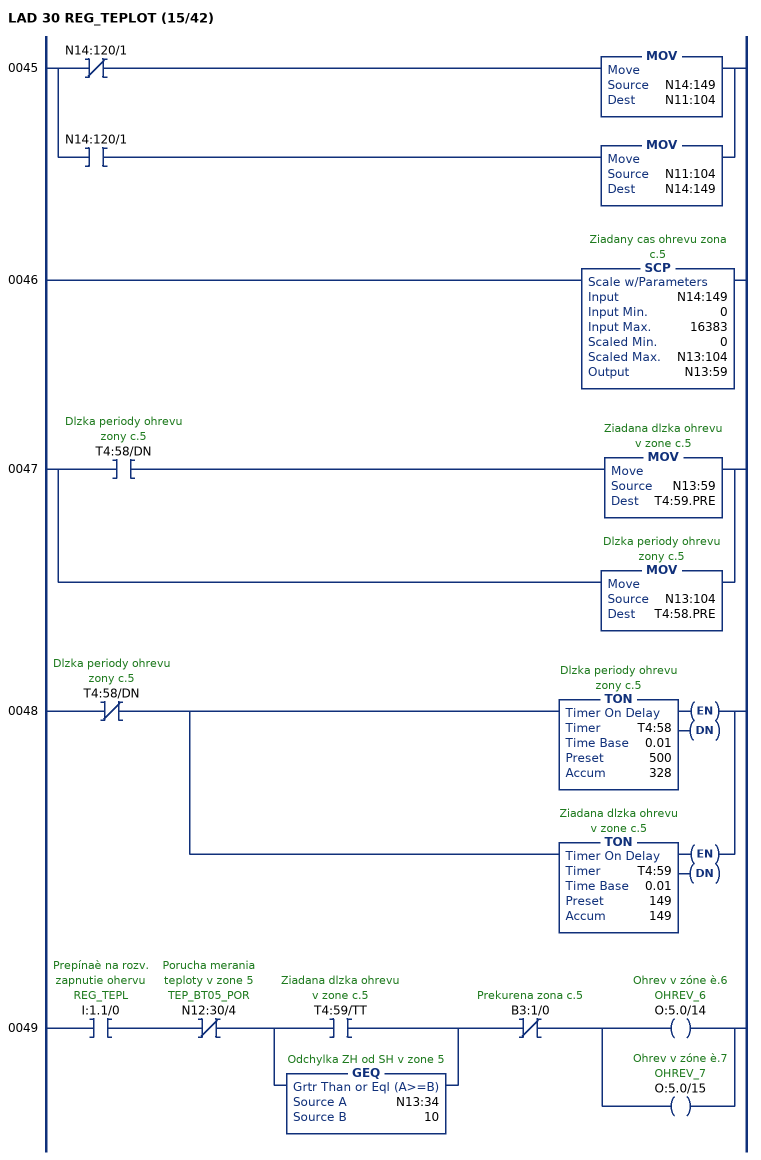
% Rung: 45 %
SOR BST XIO N14:120/1 MOV N14:149 N11:104 NXB XIC N14:120/1 MOV N11:104 N14:149 BND EOR
% Rung: 46 %
SOR SCP N14:149 0 16383 0 N13:104 N13:59 EOR
%   N13:59  "Ziadany cas ohrevu zona c.5" %
% Rung: 47 %
SOR BST XIC T4:58/DN MOV N13:59 T4:59.PRE NXB MOV N13:104 T4:58.PRE BND EOR
%   T4:58  "Dlzka periody ohrevu zony c.5" %
%   N13:59  "Ziadany cas ohrevu zona c.5" %
%   T4:59  "Ziadana dlzka ohrevu v zone c.5" %
% Rung: 48 %
SOR XIO T4:58/DN BST TON T4:58 0.01 500 328 NXB TON T4:59 0.01 149 149 BND EOR
%   T4:58  "Dlzka periody ohrevu zony c.5" %
%   T4:59  "Ziadana dlzka ohrevu v zone c.5" %
% Rung: 49 %
SOR XIC I:1.1/0 XIO N12:30/4 BST XIC T4:59/TT NXB GEQ N13:34 10 BND XIO B3:1/0 BST OTE O:5.0/14 NXB OTE O:5.0/15 BND EOR
%   I:1.1/0  REG_TEPL  "Prepínaè na rozv. zapnutie ohervu" %
%   N12:30/4  TEP_BT05_POR  "Porucha merania teploty v zone 5" %
%   T4:59  "Ziadana dlzka ohrevu v zone c.5" %
%   N13:34  "Odchylka ZH od SH v zone 5" %
%   B3:1/0  "Prekurena zona c.5" %
%   O:5.0/14  OHREV_6  "Ohrev v zóne è.6" %
%   O:5.0/15  OHREV_7  "Ohrev v zóne è.7" %

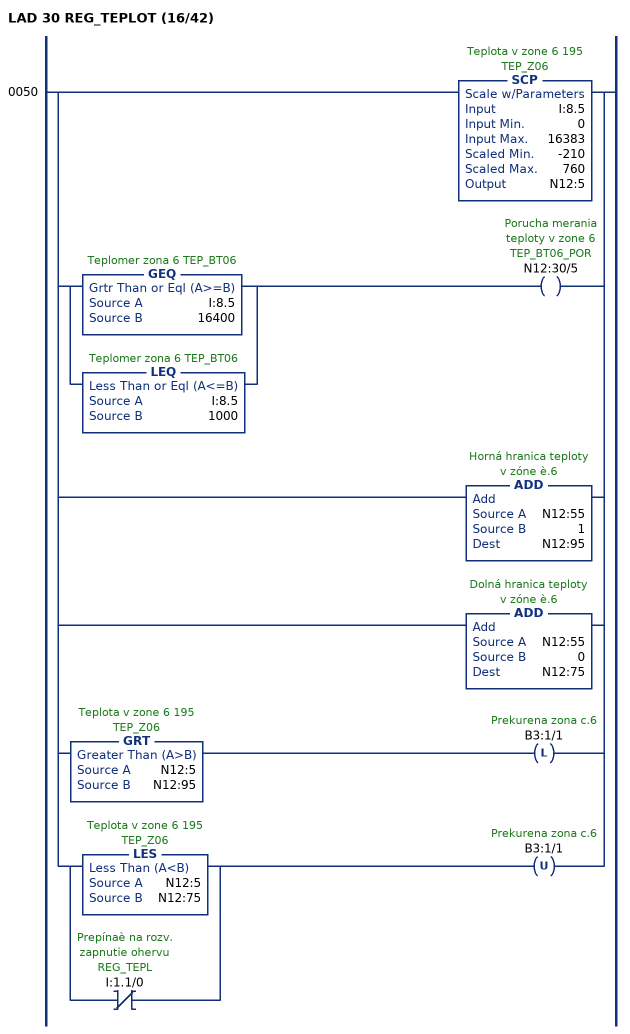
% Rung: 50 %
SOR BST SCP I:8.5 0 16383 -210 760 N12:5 NXB BST GEQ I:8.5 16400 NXB LEQ I:8.5 1000 BND OTE N12:30/5 NXB ADD N12:55 1 N12:95 NXB ADD N12:55 0 N12:75 NXB GRT N12:5 N12:95 OTL B3:1/1 NXB BST LES N12:5 N12:75 NXB XIO I:1.1/0 BND OTU B3:1/1 BND EOR
%   I:8.5  TEP_BT06  "Teplomer zona 6" %
%   N12:5  TEP_Z06  "Teplota v zone 6 195" %
%   N12:30/5  TEP_BT06_POR  "Porucha merania teploty v zone 6" %
%   N12:55  "Žiadaná teplota v zóne è.6" %
%   N12:95  "Horná hranica teploty v zóne è.6" %
%   N12:75  "Dolná hranica teploty v zóne è.6" %
%   B3:1/1  "Prekurena zona c.6" %
%   I:1.1/0  REG_TEPL  "Prepínaè na rozv. zapnutie ohervu" %

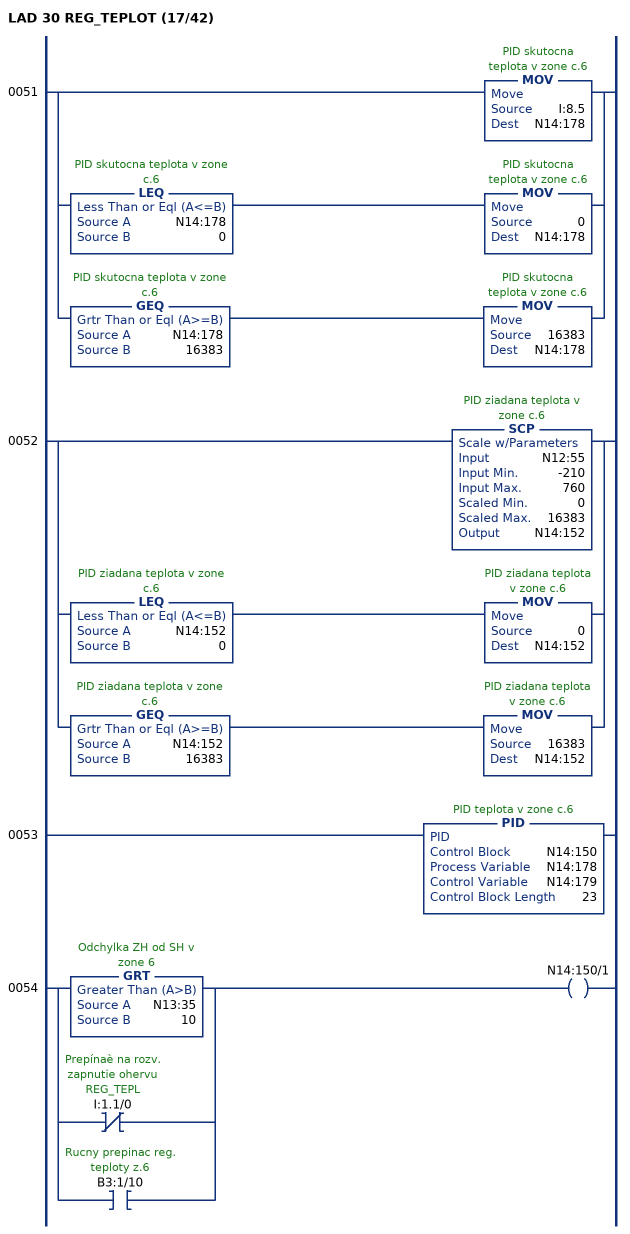
% Rung: 51 %
SOR BST MOV I:8.5 N14:178 NXB LEQ N14:178 0 MOV 0 N14:178 NXB GEQ N14:178 16383 MOV 16383 N14:178 BND EOR
%   I:8.5  TEP_BT06  "Teplomer zona 6" %
%   N14:178  "PID skutocna teplota v zone c.6" %
% Rung: 52 %
SOR BST SCP N12:55 -210 760 0 16383 N14:152 NXB LEQ N14:152 0 MOV 0 N14:152 NXB GEQ N14:152 16383 MOV 16383 N14:152 BND EOR
%   N12:55  "Žiadaná teplota v zóne è.6" %
%   N14:152  "PID ziadana teplota v zone c.6" %
% Rung: 53 %
SOR PID N14:150 N14:178 N14:179 23 EOR
%   N14:150  "PID teplota v zone c.6" %
%   N14:178  "PID skutocna teplota v zone c.6" %
% Rung: 54 %
SOR BST GRT N13:35 10 NXB XIO I:1.1/0 NXB XIC B3:1/10 BND OTE N14:150/1 EOR
%   N13:35  "Odchylka ZH od SH v zone 6" %
%   I:1.1/0  REG_TEPL  "Prepínaè na rozv. zapnutie ohervu" %
%   B3:1/10  "Rucny prepinac reg. teploty z.6" %

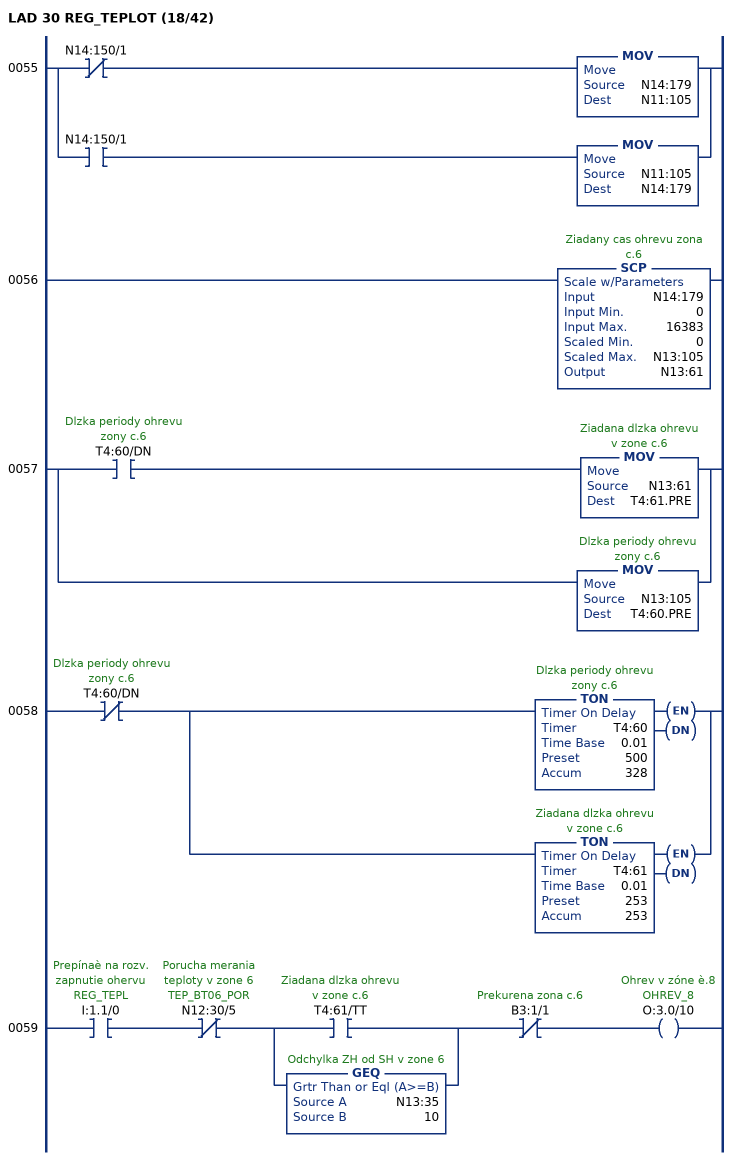
% Rung: 55 %
SOR BST XIO N14:150/1 MOV N14:179 N11:105 NXB XIC N14:150/1 MOV N11:105 N14:179 BND EOR
% Rung: 56 %
SOR SCP N14:179 0 16383 0 N13:105 N13:61 EOR
%   N13:61  "Ziadany cas ohrevu zona c.6" %
% Rung: 57 %
SOR BST XIC T4:60/DN MOV N13:61 T4:61.PRE NXB MOV N13:105 T4:60.PRE BND EOR
%   T4:60  "Dlzka periody ohrevu zony c.6" %
%   N13:61  "Ziadany cas ohrevu zona c.6" %
%   T4:61  "Ziadana dlzka ohrevu v zone c.6" %
% Rung: 58 %
SOR XIO T4:60/DN BST TON T4:60 0.01 500 328 NXB TON T4:61 0.01 253 253 BND EOR
%   T4:60  "Dlzka periody ohrevu zony c.6" %
%   T4:61  "Ziadana dlzka ohrevu v zone c.6" %
% Rung: 59 %
SOR XIC I:1.1/0 XIO N12:30/5 BST XIC T4:61/TT NXB GEQ N13:35 10 BND XIO B3:1/1 OTE O:3.0/10 EOR
%   I:1.1/0  REG_TEPL  "Prepínaè na rozv. zapnutie ohervu" %
%   N12:30/5  TEP_BT06_POR  "Porucha merania teploty v zone 6" %
%   T4:61  "Ziadana dlzka ohrevu v zone c.6" %
%   N13:35  "Odchylka ZH od SH v zone 6" %
%   B3:1/1  "Prekurena zona c.6" %
%   O:3.0/10  OHREV_8  "Ohrev v zóne è.8" %

